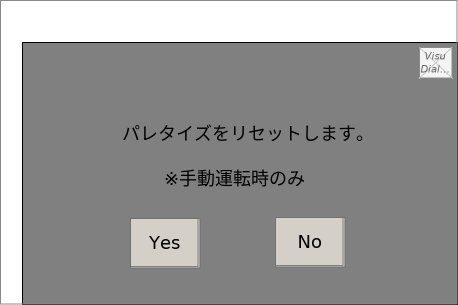
VISUALIZATION d_palletizeReset  // 458x305
    Rectangle (22,42 436x263)
    Image (419,47 33x31), image: VisuDialogs.ImagePoolDialogs.Delete
        OnMouseClick: CloseDialog Dialog=d_palletizeReset, Result=OK, NumpadKeypadSet=True
    Button (130,218 70x50), "Yes"
        tap gvl_visu.flg_btn_clrPockertQty
        OnMouseClick: CloseDialog Dialog=d_palletizeReset, Result=OK, NumpadKeypadSet=True
    Button (275,217 70x50), "No"
        OnMouseClick: CloseDialog Dialog=d_palletizeReset, Result=OK, NumpadKeypadSet=True
    Label (66,105 364x58), "パレタイズをリセットします。"
    Label (67,150 335x58), "※手動運転時のみ"
END_VISUALIZATION

(* stored: Version 1.1.0.1, ProductVersion 3.1.4024.12
   Visu d_palletizeReset: Id {7e876a85-ec85-42de-a8b2-4492556869ea} *)
